Staubli VAL3: remote_rstLight.pgx

program remote_rstLight()
begin
  // START
  if saveData:sOutStart!=""
    if inOut:dOutput[saveData:sOutStart].bActive
      inOut:dOutput[saveData:sOutStart].dDio=false
    endIf
  endIf
  // STOP
  if saveData:sOutStop!=""
    if inOut:dOutput[saveData:sOutStop].bActive
      inOut:dOutput[saveData:sOutStop].dDio=false
    endIf
  endIf
  // END
  if saveData:sOutEnd!=""
    if inOut:dOutput[saveData:sOutEnd].bActive
      inOut:dOutput[saveData:sOutEnd].dDio=false
    endIf
  endIf
  // HOME
  if saveData:sOutHome!=""
    if inOut:dOutput[saveData:sOutHome].bActive
      inOut:dOutput[saveData:sOutHome].dDio=false
    endIf
  endIf
end
